// SIMATIC S7-200 project (STEP 7-Micro/WIN), CPU 226 CN REL 02.01

SYMBOL_TABLE 用户定义1
Write_Output_Done M2.3     // 写从站实际输出值完成位
Read_Inputs_Done M2.2     // 读取从站输入点完成位
Read_Register_Done M2.1     // 读保存寄存器完成位
Start_MBUS_MSG   M0.1     // 初始化完成，启动读/写功能
MBUS_CTRL_Error  MB1      // Modbus主站初始化错误代码
MBUS_CTRL_Done   M0.0     // Modbus主站初始化完成位
END_SYMBOL_TABLE

SYMBOL_TABLE S7-200 符号
Always_On        SM0.0    // 始终接通为 ON
First_Scan_On    SM0.1    // 仅第一个扫描周期中接通为 ON
END_SYMBOL_TABLE

ORGANIZATION_BLOCK 主程序:OB1
TITLE=系统启动时，当首次扫描标志为1，PLC复位Modbus主站初始化完成标志，确保系统从干净状态开始。接着，PLC调用子程序，以始终接通标志驱动初始化，设置波特率为9600、无奇偶校验、超时时间1000ms，并通过Modbus主站初始化完成标志确认初始化成功——只有在初始化成功后，Modbus主站初始化完成标志才会置1，否则Modbus主站初始化错误代码会记录错误原因，如波特率无效。
// 
// 初始化完成后，PLC利用Modbus主站读写请求位和定时器定期触发读写操作。当Modbus主站初始化完成标志为1时，置位Modbus主站读写请求位，启动读写功能。同时，定时器在始终接通标志驱动下，每15个时间单位触发一次，置位定时器触发标志，确保系统定期从从站读取数据，防止长时间无通信导致监控失效。读取操作通过调用子程序实现，从从站地址为1的保持寄存器读取13个字的数据（如温度和压力值），并将数据存入保持寄存器数据缓冲区。操作完成后，Modbus读保持寄存器完成位置1，并复位Modbus主站读写请求位和定时器触发标志，以便下一次操作——即每次读取操作完成后，系统会自动准备下一次读取。
// 
// 在整个过程中，保持寄存器数据缓冲区必须正确配置，连续存储13个字的数据，确保温度和压力值的准确存储和访问。此外，系统通过检查Modbus主站初始化错误代码和Modbus读写错误代码来处理可能出现的通讯错误，例如从站无响应或校验错误——只有当错误代码为0时，数据才被认为是可靠的。通过这种设计，PLC能够可靠地与从站设备通信，实时读取温度和压力数据并为后续控制提供依据。
BEGIN
Network 1
// 第一扫秒周期, 复位各标志位和起始位
LD     First_Scan_On:SM0.1
R      MBUS_CTRL_Done:M0.0, 2
?000
Network 2
// Modbus 主站初始化完成后, 启动读写指令
LD     MBUS_CTRL_Done:M0.0
EU
S      Start_MBUS_MSG:M0.1, 1
Network 3
LD     Always_On:SM0.0
AN     M0.2
TON    T40, 15
Network 4
LD     T40
=      M0.2
Network 5 // 网络标题
//       
LD     Always_On:SM0.0
=      L60.0
LD     Always_On:SM0.0
=      L63.7
LD     L60.0
CALL   MBUS_CTRL:SBR1, L63.7, 9600, 0, 1000, MBUS_CTRL_Done:M0.0, MBUS_CTRL_Error:MB1
Network 6
// 读取从站保持寄存器的数据
LD     Start_MBUS_MSG:M0.1
O      M0.2
=      L60.0
LD     Start_MBUS_MSG:M0.1
EU
LD     M0.2
EU
OLD
=      L63.7
LD     L60.0
CALL   MBUS_MSG:SBR2, L63.7, 1, 0, 40002, 13, &VB1000, Read_Register_Done:M2.1, MB2
Network 7
// 读取从站保持寄存器的数据完成，复位请求
LD     Read_Register_Done:M2.1
R      Start_MBUS_MSG:M0.1, 1
R      M0.2, 1
Network 8
LD     Always_On:SM0.0
MOVW   VW1000, VW1000
MOVW   VW1002, VW1002
MOVW   VW1004, VW1004
MOVW   VW1006, VW1006
MOVW   VW1008, VW1008
MOVW   VW1010, VW1010
MOVW   VW1018, VW1018
MOVW   VW1020, VW1020
MOVW   VW1022, VW1022
MOVW   VW1024, VW1024
END_ORGANIZATION_BLOCK

// SBR1: protected block, not included

// SBR2: protected block, not included

// SBR3: protected block, not included
